{attribute 'reflection'} 
FUNCTION_BLOCK FB_LAMP_ONOFF IMPLEMENTS I_Lamp
VAR	
	// Hardware control variables
	bOutHw AT %Q*:BOOL;
	
	// Instance-path variable
    {attribute 'instance-path'} 
    {attribute 'noinit'} 
    sPath : STRING; 
END_VAR

METHOD OFF : BOOL
bOutHw := FALSE;
END_METHOD

METHOD ON : BOOL
bOutHw := TRUE;
END_METHOD

PROPERTY State : STRING
GET
State := CONCAT('Object: ', sPath);
State := CONCAT(State, ' State:');
State := CONCAT(State, BOOL_TO_STRING(THIS^.bOutHw));
END_GET
END_PROPERTY

END_FUNCTION_BLOCK

(* stored: Version 1.1.0.1, ProductVersion 3.1.4024.6
   POU FB_LAMP_ONOFF: Id {aa995fee-1421-4b66-801f-824f527031c6}, SpecialFunc None
   Method OFF: Id {604fc7c4-a3e8-4532-885f-37030c4716a7}
   Method ON: Id {bab13569-3551-452d-8fd5-968e8f0ea75b}
   Property State: Id {c6c150c1-88e5-42cd-91a3-2cbe3b0c34c9}
   Get Get: Id {7331da31-b73b-4569-afea-cbe7125fd6f3} *)
